{attribute 'GeneratedUsingTerminal: EL3255-0000-0016'}
{attribute addProperty BoxType "EL3255-0000-0016"}
{attribute addProperty Description "EL3255 5Ch. potentiometer measurement with sensor supply"}
{attribute addProperty Physics "KK"}
{attribute addProperty Id "RTD_Standard_Channel_1AT %I*RTD_Standard_Channel_A8DF64E310RTD_Standard_Channel_2AT %I*RTD_Standard_Channel_A8DF64E310RTD_Standard_Channel_3AT %I*RTD_Standard_Channel_A8DF64E310RTD_Standard_Channel_4AT %I*RTD_Standard_Channel_A8DF64E310RTD_Standard_Channel_5AT %I*RTD_Standard_Channel_A8DF64E310WcStateAT %I*WcState_9091E0EB2InfoDataAT %I*InfoData_32EB74EA10"}
{attribute addProperty CRC "1885800497"}
{attribute addProperty Size "62"}
TYPE EL3255_70670831 EXTENDS EtcSlaveTerminalBase_947E5A46 :
STRUCT
	{attribute addProperty Name "RTD_Standard_Channel_1"}
	RTD_Standard_Channel_1 : RTD_Standard_Channel_A8DF64E3;
	{attribute addProperty Name "RTD_Standard_Channel_2"}
	RTD_Standard_Channel_2 : RTD_Standard_Channel_A8DF64E3;
	{attribute addProperty Name "RTD_Standard_Channel_3"}
	RTD_Standard_Channel_3 : RTD_Standard_Channel_A8DF64E3;
	{attribute addProperty Name "RTD_Standard_Channel_4"}
	RTD_Standard_Channel_4 : RTD_Standard_Channel_A8DF64E3;
	{attribute addProperty Name "RTD_Standard_Channel_5"}
	RTD_Standard_Channel_5 : RTD_Standard_Channel_A8DF64E3;
	{attribute addProperty Name "WcState"}
	WcState : WcState_9091E0EB;
	{attribute addProperty Name "InfoData"}
	InfoData : InfoData_32EB74EA;
END_STRUCT
END_TYPE

(* stored: Version 1.2.0.0, ProductVersion 3.1.4024.11
   DUT EL3255_70670831: Id {0188b944-4ea6-403e-acb2-47d8c67ebeee} *)
